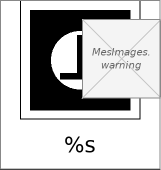
VISUALIZATION VISU_POMPE_ROOTS  // 161x170
VAR_IN_OUT
	m_Input_POMPE : BLOCK_PPM;
END_VAR
    Rectangle (0,0 160x170), invisible if: TRUE
    Rectangle (10,130 140x30), "%s", text variable: m_Input_POMPE.MNEMO
    Rectangle (30,10 100x100)
    Rectangle (30,10 100x100), colour toggle: (m_Input_POMPE.STATE_ON) <> 0, invisible if: NOT m_Input_POMPE.STATE_ON AND NOT m_Input_POMPE.STATE_OFF
    Ellipse (46,26 68x68)
    Rectangle (20,0 120x119), invisible if: NOT (m_Input_POMPE.Autor_ON_IHM OR m_Input_POMPE.Autor_OFF_IHM) OR NOT PRG_User.ACTU_USER.MAINTENANCE
        tap m_Input_POMPE.M_ON
    Rectangle (77,35 6x39)
    Rectangle (60,73 41x6)
    Image (82,19 79x79), invisible if: NOT m_Input_POMPE.STATE_NOK, image: MesImages.warning
END_VISUALIZATION

(* stored: Version 1.1.0.1, ProductVersion 3.1.4024.10
   Visu VISU_POMPE_ROOTS: Id {ffaf5462-586e-44b8-b6ea-25a445a8cc3d} *)
